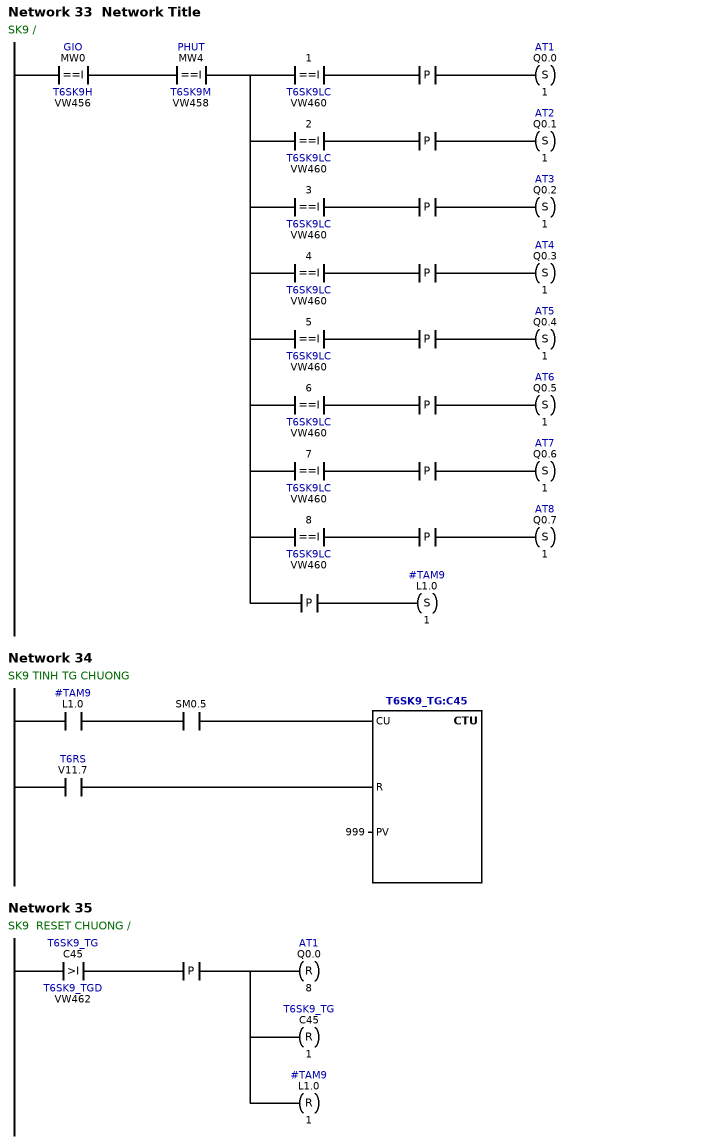
[picture p48: SBR7 networks 33-35]
Network 33 // Network Title
// SK9
// 	
LDW=   GIO:MW0, T6SK9H:VW456
AW=    PHUT:MW4, T6SK9M:VW458
LPS
AW=    1, T6SK9LC:VW460
EU
S      AT1:Q0.0, 1
LRD
AW=    2, T6SK9LC:VW460
EU
S      AT2:Q0.1, 1
LRD
AW=    3, T6SK9LC:VW460
EU
S      AT3:Q0.2, 1
LRD
AW=    4, T6SK9LC:VW460
EU
S      AT4:Q0.3, 1
LRD
AW=    5, T6SK9LC:VW460
EU
S      AT5:Q0.4, 1
LRD
AW=    6, T6SK9LC:VW460
EU
S      AT6:Q0.5, 1
LRD
AW=    7, T6SK9LC:VW460
EU
S      AT7:Q0.6, 1
LRD
AW=    8, T6SK9LC:VW460
EU
S      AT8:Q0.7, 1
LPP
EU
S      #TAM9:L1.0, 1
Network 34
// SK9 TINH TG CHUONG
LD     #TAM9:L1.0
A      SM0.5
LD     T6RS:V11.7
CTU    T6SK9_TG:C45, 999
Network 35
// SK9  RESET CHUONG
// 
LDW>   T6SK9_TG:C45, T6SK9_TGD:VW462
EU
R      AT1:Q0.0, 8
R      T6SK9_TG:C45, 1
R      #TAM9:L1.0, 1
Network 44 // Network Title
// Network Comment
Network 54 // Network Title
// Network Comment
Network 64 // Network Title
// Network Comment
Network 74 // Network Title
// Network Comment
END_SUBROUTINE_BLOCK

SUBROUTINE_BLOCK TH7:SBR8
TITLE=SUBROUTINE COMMENTS
VAR
TAM1:BOOL;	// L0.0 
TAM2:BOOL;	// L0.1 
TAM3:BOOL;	// L0.2 
TAM4:BOOL;	// L0.3 
TAM5:BOOL;	// L0.4 
TAM6:BOOL;	// L0.5 
TAM7:BOOL;	// L0.6 
TAM8:BOOL;	// L0.7 
TAM9:BOOL;	// L1.0 
END_VAR
BEGIN
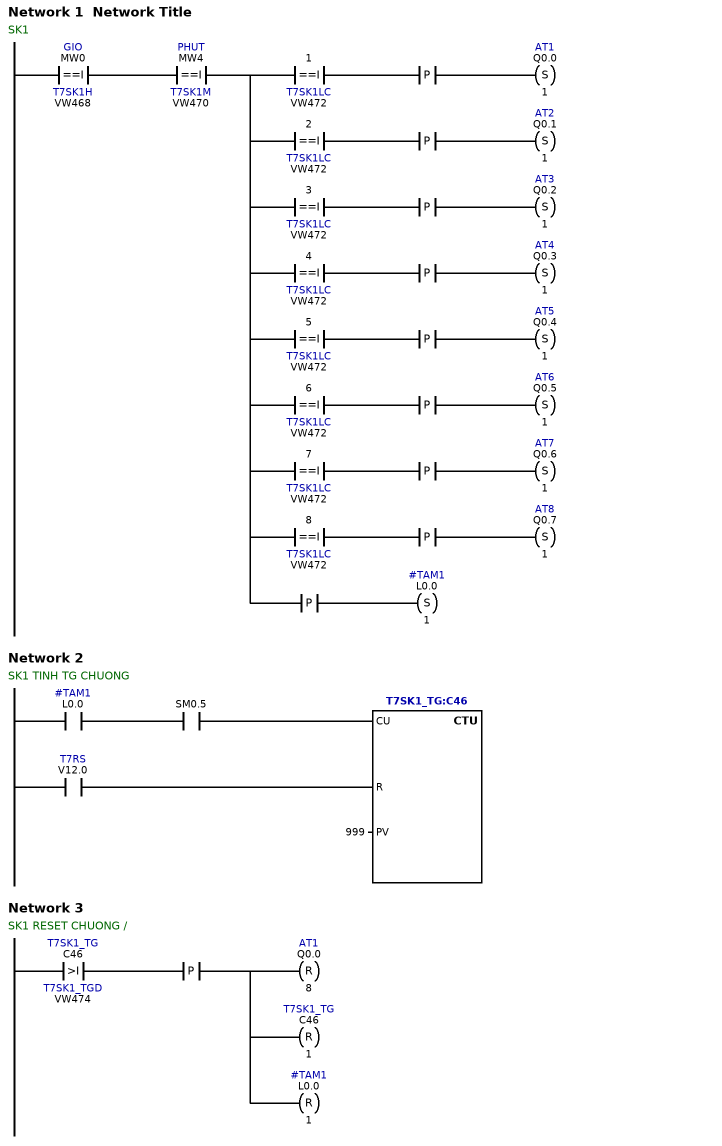
Network 1 // Network Title
// SK1	
LDW=   GIO:MW0, T7SK1H:VW468
AW=    PHUT:MW4, T7SK1M:VW470
LPS
AW=    1, T7SK1LC:VW472
EU
S      AT1:Q0.0, 1
LRD
AW=    2, T7SK1LC:VW472
EU
S      AT2:Q0.1, 1
LRD
AW=    3, T7SK1LC:VW472
EU
S      AT3:Q0.2, 1
LRD
AW=    4, T7SK1LC:VW472
EU
S      AT4:Q0.3, 1
LRD
AW=    5, T7SK1LC:VW472
EU
S      AT5:Q0.4, 1
LRD
AW=    6, T7SK1LC:VW472
EU
S      AT6:Q0.5, 1
LRD
AW=    7, T7SK1LC:VW472
EU
S      AT7:Q0.6, 1
LRD
AW=    8, T7SK1LC:VW472
EU
S      AT8:Q0.7, 1
LPP
EU
S      #TAM1:L0.0, 1
Network 2
// SK1 TINH TG CHUONG
LD     #TAM1:L0.0
A      SM0.5
LD     T7RS:V12.0
CTU    T7SK1_TG:C46, 999
Network 3
// SK1 RESET CHUONG
// 
LDW>   T7SK1_TG:C46, T7SK1_TGD:VW474
EU
R      AT1:Q0.0, 8
R      T7SK1_TG:C46, 1
R      #TAM1:L0.0, 1
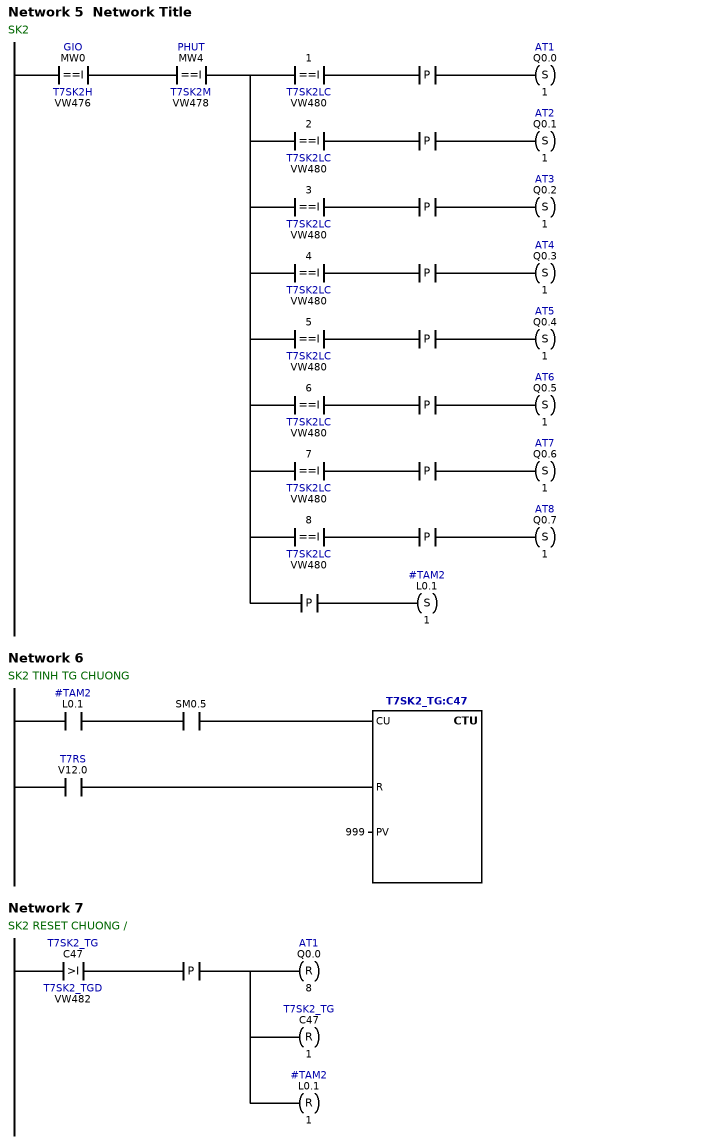
Network 5 // Network Title
// SK2
LDW=   GIO:MW0, T7SK2H:VW476
AW=    PHUT:MW4, T7SK2M:VW478
LPS
AW=    1, T7SK2LC:VW480
EU
S      AT1:Q0.0, 1
LRD
AW=    2, T7SK2LC:VW480
EU
S      AT2:Q0.1, 1
LRD
AW=    3, T7SK2LC:VW480
EU
S      AT3:Q0.2, 1
LRD
AW=    4, T7SK2LC:VW480
EU
S      AT4:Q0.3, 1
LRD
AW=    5, T7SK2LC:VW480
EU
S      AT5:Q0.4, 1
LRD
AW=    6, T7SK2LC:VW480
EU
S      AT6:Q0.5, 1
LRD
AW=    7, T7SK2LC:VW480
EU
S      AT7:Q0.6, 1
LRD
AW=    8, T7SK2LC:VW480
EU
S      AT8:Q0.7, 1
LPP
EU
S      #TAM2:L0.1, 1
Network 6
// SK2 TINH TG CHUONG
LD     #TAM2:L0.1
A      SM0.5
LD     T7RS:V12.0
CTU    T7SK2_TG:C47, 999
Network 7
// SK2 RESET CHUONG
// 
LDW>   T7SK2_TG:C47, T7SK2_TGD:VW482
EU
R      AT1:Q0.0, 8
R      T7SK2_TG:C47, 1
R      #TAM2:L0.1, 1
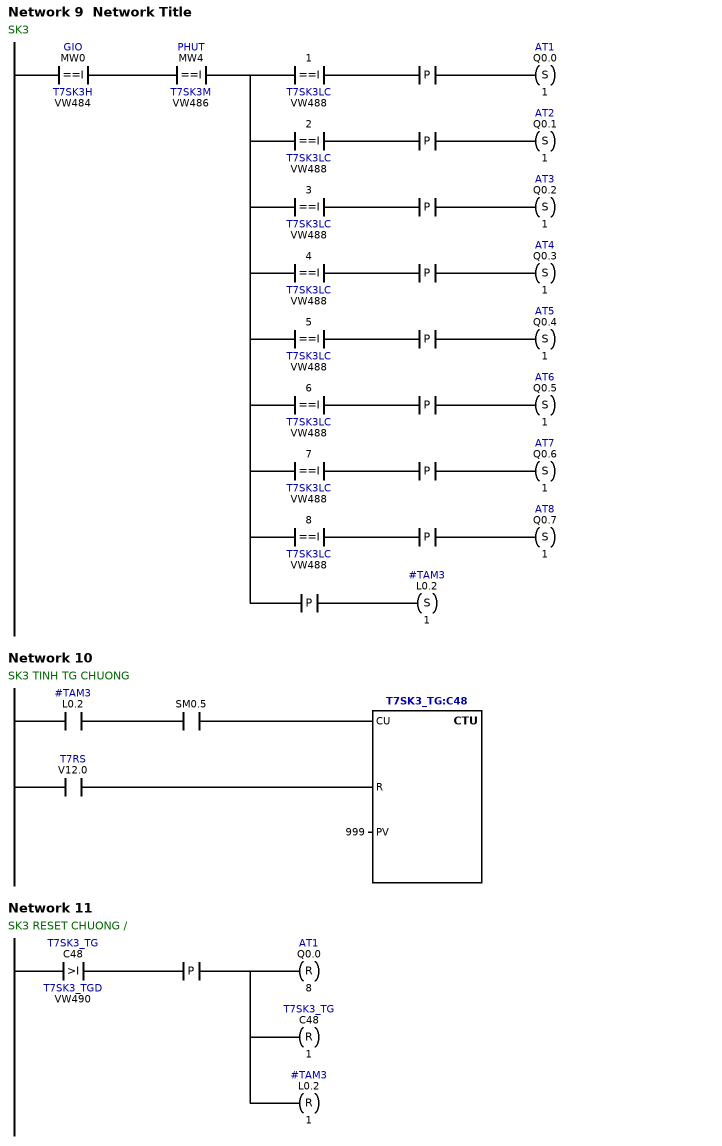
Network 9 // Network Title
// SK3	
LDW=   GIO:MW0, T7SK3H:VW484
AW=    PHUT:MW4, T7SK3M:VW486
LPS
AW=    1, T7SK3LC:VW488
EU
S      AT1:Q0.0, 1
LRD
AW=    2, T7SK3LC:VW488
EU
S      AT2:Q0.1, 1
LRD
AW=    3, T7SK3LC:VW488
EU
S      AT3:Q0.2, 1
LRD
AW=    4, T7SK3LC:VW488
EU
S      AT4:Q0.3, 1
LRD
AW=    5, T7SK3LC:VW488
EU
S      AT5:Q0.4, 1
LRD
AW=    6, T7SK3LC:VW488
EU
S      AT6:Q0.5, 1
LRD
AW=    7, T7SK3LC:VW488
EU
S      AT7:Q0.6, 1
LRD
AW=    8, T7SK3LC:VW488
EU
S      AT8:Q0.7, 1
LPP
EU
S      #TAM3:L0.2, 1
Network 10
// SK3 TINH TG CHUONG
LD     #TAM3:L0.2
A      SM0.5
LD     T7RS:V12.0
CTU    T7SK3_TG:C48, 999
Network 11
// SK3 RESET CHUONG
// 
LDW>   T7SK3_TG:C48, T7SK3_TGD:VW490
EU
R      AT1:Q0.0, 8
R      T7SK3_TG:C48, 1
R      #TAM3:L0.2, 1
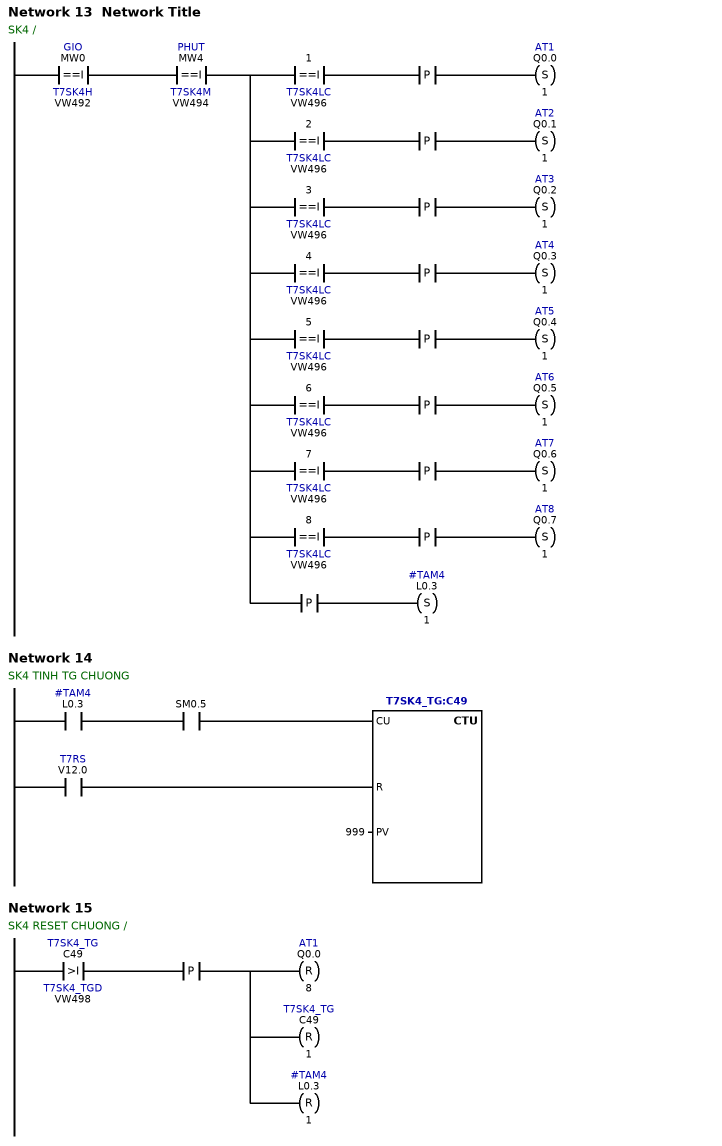
Network 13 // Network Title
// SK4
// 	
LDW=   GIO:MW0, T7SK4H:VW492
AW=    PHUT:MW4, T7SK4M:VW494
LPS
AW=    1, T7SK4LC:VW496
EU
S      AT1:Q0.0, 1
LRD
AW=    2, T7SK4LC:VW496
EU
S      AT2:Q0.1, 1
LRD
AW=    3, T7SK4LC:VW496
EU
S      AT3:Q0.2, 1
LRD
AW=    4, T7SK4LC:VW496
EU
S      AT4:Q0.3, 1
LRD
AW=    5, T7SK4LC:VW496
EU
S      AT5:Q0.4, 1
LRD
AW=    6, T7SK4LC:VW496
EU
S      AT6:Q0.5, 1
LRD
AW=    7, T7SK4LC:VW496
EU
S      AT7:Q0.6, 1
LRD
AW=    8, T7SK4LC:VW496
EU
S      AT8:Q0.7, 1
LPP
EU
S      #TAM4:L0.3, 1
Network 14
// SK4 TINH TG CHUONG
LD     #TAM4:L0.3
A      SM0.5
LD     T7RS:V12.0
CTU    T7SK4_TG:C49, 999
Network 15
// SK4 RESET CHUONG
// 
LDW>   T7SK4_TG:C49, T7SK4_TGD:VW498
EU
R      AT1:Q0.0, 8
R      T7SK4_TG:C49, 1
R      #TAM4:L0.3, 1
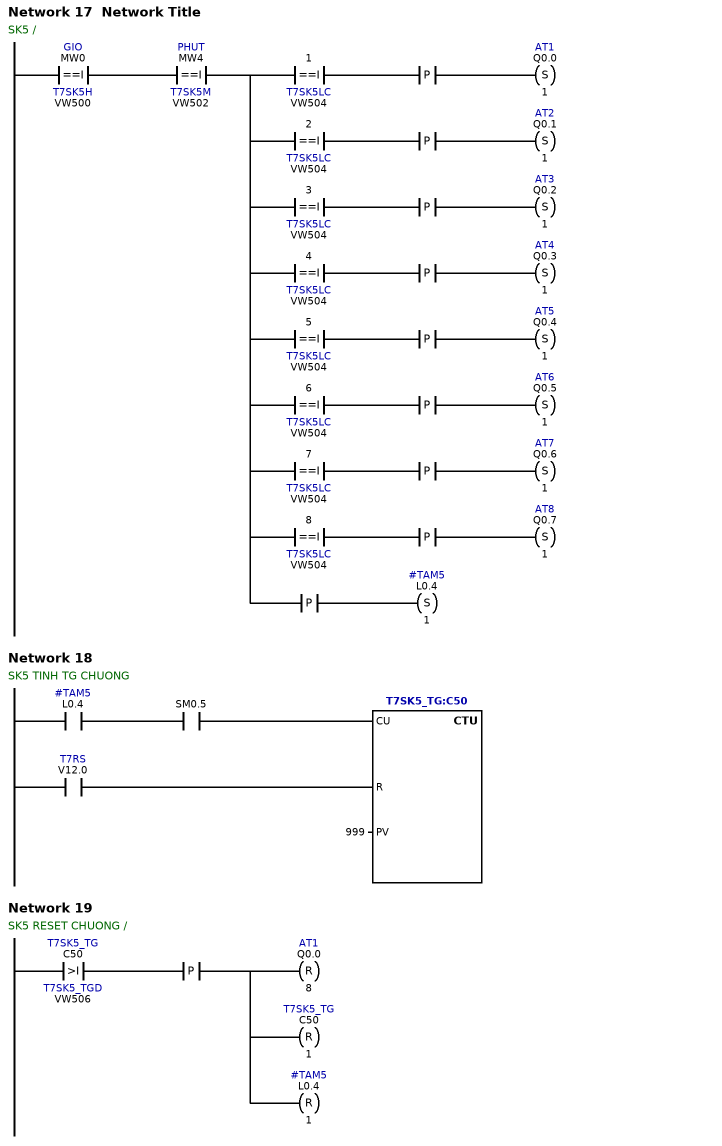
Network 17 // Network Title
// SK5
// 	
LDW=   GIO:MW0, T7SK5H:VW500
AW=    PHUT:MW4, T7SK5M:VW502
LPS
AW=    1, T7SK5LC:VW504
EU
S      AT1:Q0.0, 1
LRD
AW=    2, T7SK5LC:VW504
EU
S      AT2:Q0.1, 1
LRD
AW=    3, T7SK5LC:VW504
EU
S      AT3:Q0.2, 1
LRD
AW=    4, T7SK5LC:VW504
EU
S      AT4:Q0.3, 1
LRD
AW=    5, T7SK5LC:VW504
EU
S      AT5:Q0.4, 1
LRD
AW=    6, T7SK5LC:VW504
EU
S      AT6:Q0.5, 1
LRD
AW=    7, T7SK5LC:VW504
EU
S      AT7:Q0.6, 1
LRD
AW=    8, T7SK5LC:VW504
EU
S      AT8:Q0.7, 1
LPP
EU
S      #TAM5:L0.4, 1
Network 18
// SK5 TINH TG CHUONG
LD     #TAM5:L0.4
A      SM0.5
LD     T7RS:V12.0
CTU    T7SK5_TG:C50, 999
Network 19
// SK5 RESET CHUONG
// 
LDW>   T7SK5_TG:C50, T7SK5_TGD:VW506
EU
R      AT1:Q0.0, 8
R      T7SK5_TG:C50, 1
R      #TAM5:L0.4, 1
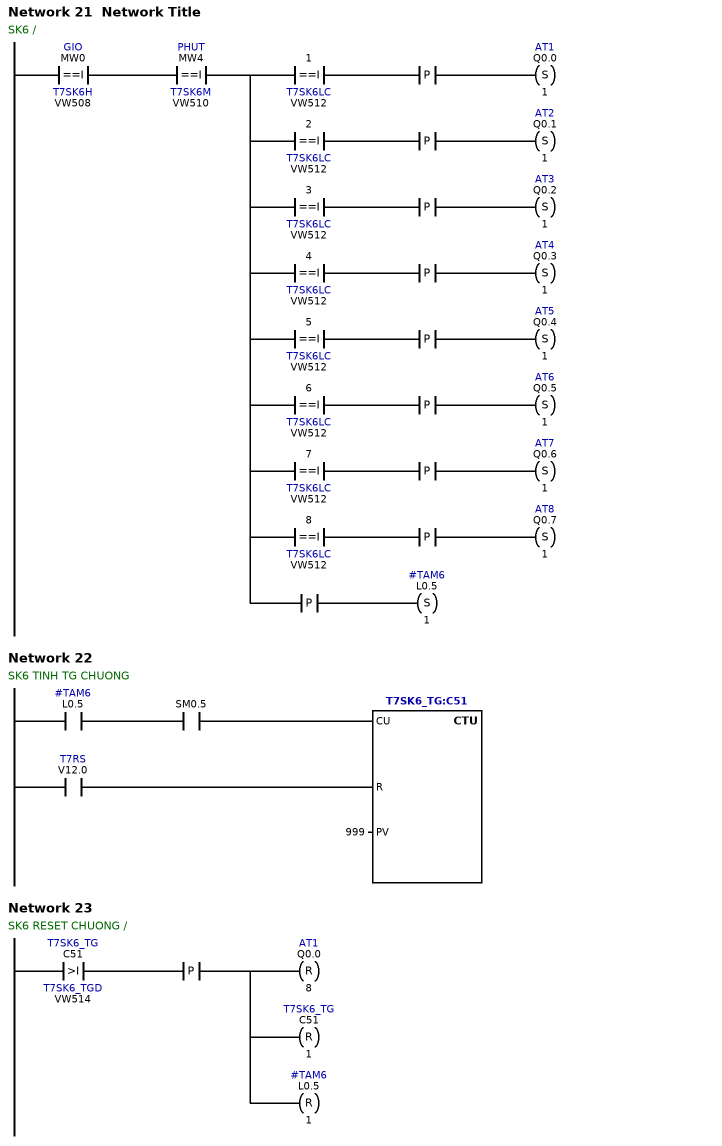
Network 21 // Network Title
// SK6
// 	
LDW=   GIO:MW0, T7SK6H:VW508
AW=    PHUT:MW4, T7SK6M:VW510
LPS
AW=    1, T7SK6LC:VW512
EU
S      AT1:Q0.0, 1
LRD
AW=    2, T7SK6LC:VW512
EU
S      AT2:Q0.1, 1
LRD
AW=    3, T7SK6LC:VW512
EU
S      AT3:Q0.2, 1
LRD
AW=    4, T7SK6LC:VW512
EU
S      AT4:Q0.3, 1
LRD
AW=    5, T7SK6LC:VW512
EU
S      AT5:Q0.4, 1
LRD
AW=    6, T7SK6LC:VW512
EU
S      AT6:Q0.5, 1
LRD
AW=    7, T7SK6LC:VW512
EU
S      AT7:Q0.6, 1
LRD
AW=    8, T7SK6LC:VW512
EU
S      AT8:Q0.7, 1
LPP
EU
S      #TAM6:L0.5, 1
Network 22
// SK6 TINH TG CHUONG
LD     #TAM6:L0.5
A      SM0.5
LD     T7RS:V12.0
CTU    T7SK6_TG:C51, 999
Network 23
// SK6 RESET CHUONG
// 
LDW>   T7SK6_TG:C51, T7SK6_TGD:VW514
EU
R      AT1:Q0.0, 8
R      T7SK6_TG:C51, 1
R      #TAM6:L0.5, 1
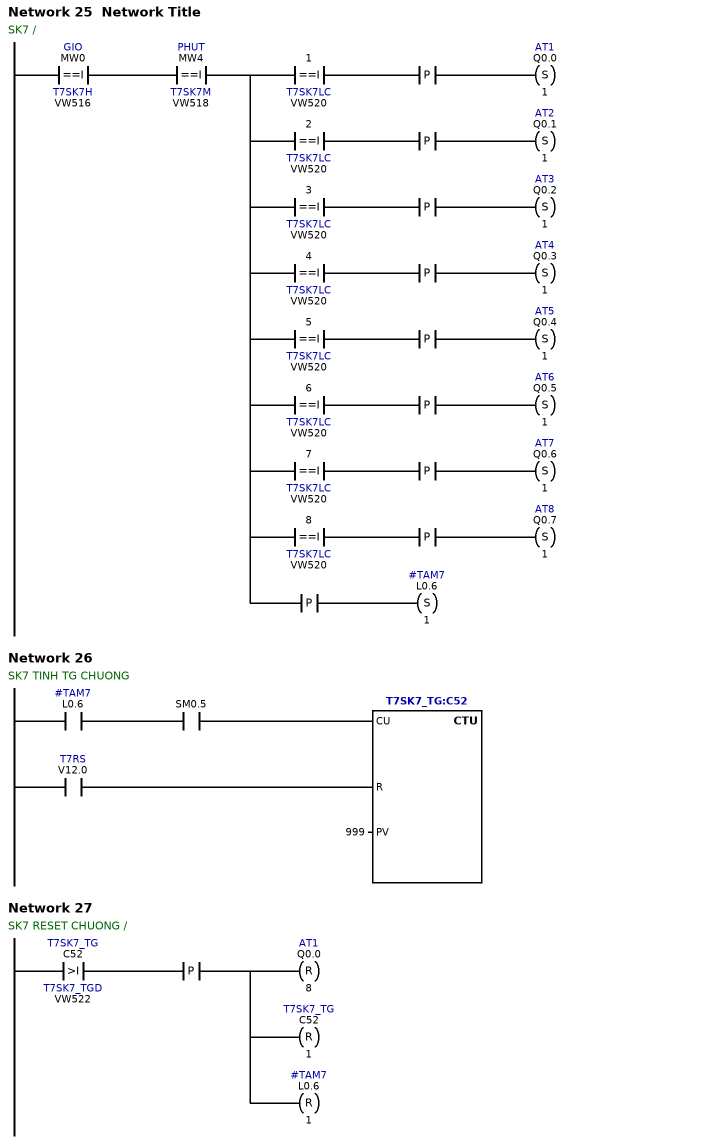
Network 25 // Network Title
// SK7
// 	
LDW=   GIO:MW0, T7SK7H:VW516
AW=    PHUT:MW4, T7SK7M:VW518
LPS
AW=    1, T7SK7LC:VW520
EU
S      AT1:Q0.0, 1
LRD
AW=    2, T7SK7LC:VW520
EU
S      AT2:Q0.1, 1
LRD
AW=    3, T7SK7LC:VW520
EU
S      AT3:Q0.2, 1
LRD
AW=    4, T7SK7LC:VW520
EU
S      AT4:Q0.3, 1
LRD
AW=    5, T7SK7LC:VW520
EU
S      AT5:Q0.4, 1
LRD
AW=    6, T7SK7LC:VW520
EU
S      AT6:Q0.5, 1
LRD
AW=    7, T7SK7LC:VW520
EU
S      AT7:Q0.6, 1
LRD
AW=    8, T7SK7LC:VW520
EU
S      AT8:Q0.7, 1
LPP
EU
S      #TAM7:L0.6, 1
Network 26
// SK7 TINH TG CHUONG
LD     #TAM7:L0.6
A      SM0.5
LD     T7RS:V12.0
CTU    T7SK7_TG:C52, 999
Network 27
// SK7 RESET CHUONG
// 
LDW>   T7SK7_TG:C52, T7SK7_TGD:VW522
EU
R      AT1:Q0.0, 8
R      T7SK7_TG:C52, 1
R      #TAM7:L0.6, 1
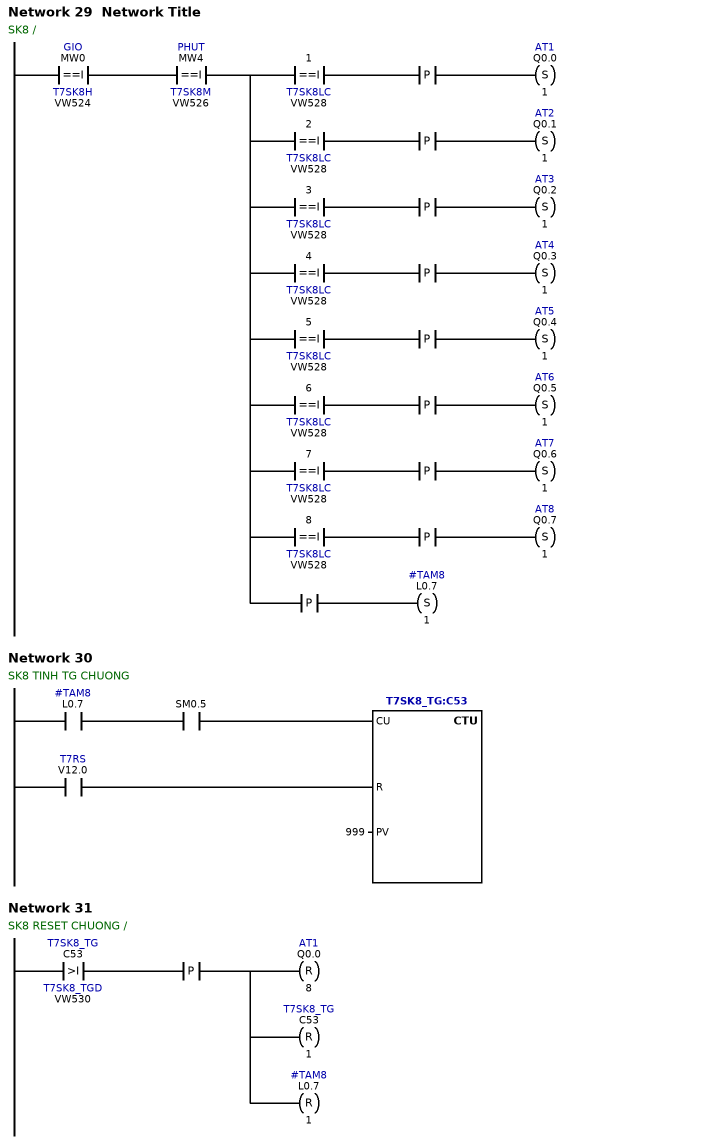
Network 29 // Network Title
// SK8
// 	
LDW=   GIO:MW0, T7SK8H:VW524
AW=    PHUT:MW4, T7SK8M:VW526
LPS
AW=    1, T7SK8LC:VW528
EU
S      AT1:Q0.0, 1
LRD
AW=    2, T7SK8LC:VW528
EU
S      AT2:Q0.1, 1
LRD
AW=    3, T7SK8LC:VW528
EU
S      AT3:Q0.2, 1
LRD
AW=    4, T7SK8LC:VW528
EU
S      AT4:Q0.3, 1
LRD
AW=    5, T7SK8LC:VW528
EU
S      AT5:Q0.4, 1
LRD
AW=    6, T7SK8LC:VW528
EU
S      AT6:Q0.5, 1
LRD
AW=    7, T7SK8LC:VW528
EU
S      AT7:Q0.6, 1
LRD
AW=    8, T7SK8LC:VW528
EU
S      AT8:Q0.7, 1
LPP
EU
S      #TAM8:L0.7, 1
Network 30
// SK8 TINH TG CHUONG
LD     #TAM8:L0.7
A      SM0.5
LD     T7RS:V12.0
CTU    T7SK8_TG:C53, 999
Network 31
// SK8 RESET CHUONG
// 
LDW>   T7SK8_TG:C53, T7SK8_TGD:VW530
EU
R      AT1:Q0.0, 8
R      T7SK8_TG:C53, 1
R      #TAM8:L0.7, 1
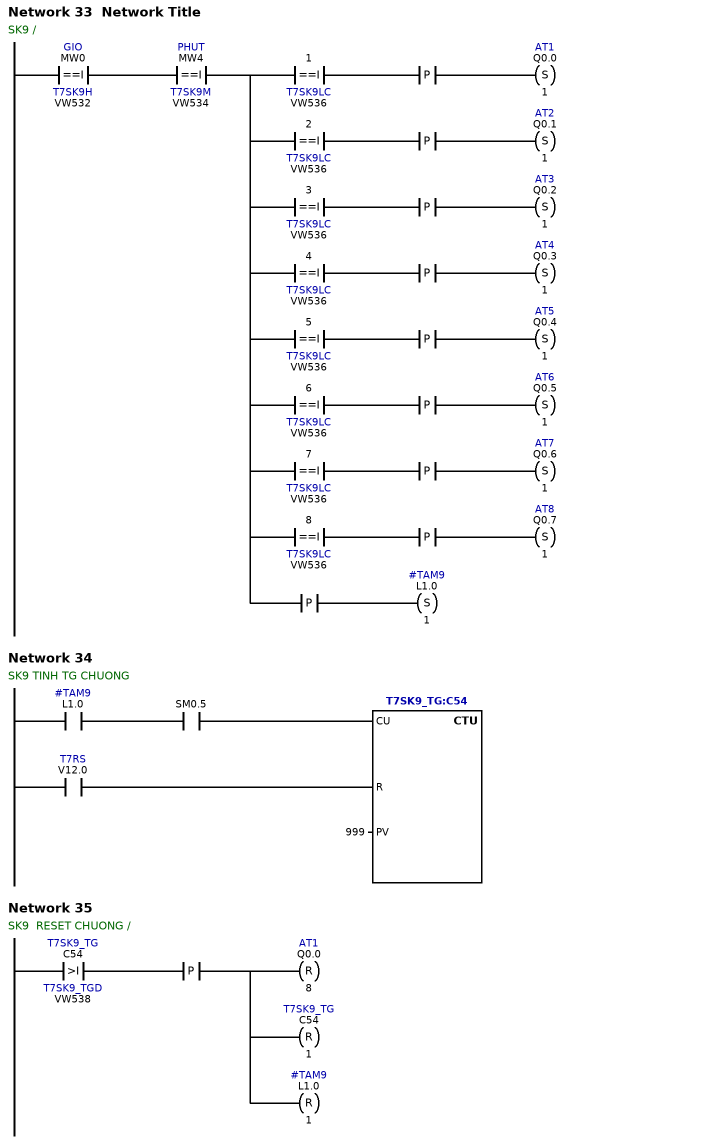
Network 33 // Network Title
// SK9
// 	
LDW=   GIO:MW0, T7SK9H:VW532
AW=    PHUT:MW4, T7SK9M:VW534
LPS
AW=    1, T7SK9LC:VW536
EU
S      AT1:Q0.0, 1
LRD
AW=    2, T7SK9LC:VW536
EU
S      AT2:Q0.1, 1
LRD
AW=    3, T7SK9LC:VW536
EU
S      AT3:Q0.2, 1
LRD
AW=    4, T7SK9LC:VW536
EU
S      AT4:Q0.3, 1
LRD
AW=    5, T7SK9LC:VW536
EU
S      AT5:Q0.4, 1
LRD
AW=    6, T7SK9LC:VW536
EU
S      AT6:Q0.5, 1
LRD
AW=    7, T7SK9LC:VW536
EU
S      AT7:Q0.6, 1
LRD
AW=    8, T7SK9LC:VW536
EU
S      AT8:Q0.7, 1
LPP
EU
S      #TAM9:L1.0, 1
Network 34
// SK9 TINH TG CHUONG
LD     #TAM9:L1.0
A      SM0.5
LD     T7RS:V12.0
CTU    T7SK9_TG:C54, 999
Network 35
// SK9  RESET CHUONG
// 
LDW>   T7SK9_TG:C54, T7SK9_TGD:VW538
EU
R      AT1:Q0.0, 8
R      T7SK9_TG:C54, 1
R      #TAM9:L1.0, 1
Network 44 // Network Title
// Network Comment
Network 54 // Network Title
// Network Comment
Network 64 // Network Title
// Network Comment
Network 74 // Network Title
// Network Comment
Network 84 // Network Title
// Network Comment
END_SUBROUTINE_BLOCK

SUBROUTINE_BLOCK CN:SBR9
TITLE=SUBROUTINE COMMENTS
VAR
TAM1:BOOL;	// L0.0 
TAM2:BOOL;	// L0.1 
TAM3:BOOL;	// L0.2 
TAM4:BOOL;	// L0.3 
TAM5:BOOL;	// L0.4 
TAM6:BOOL;	// L0.5 
TAM7:BOOL;	// L0.6 
TAM8:BOOL;	// L0.7 
TAM9:BOOL;	// L1.0 
END_VAR
BEGIN
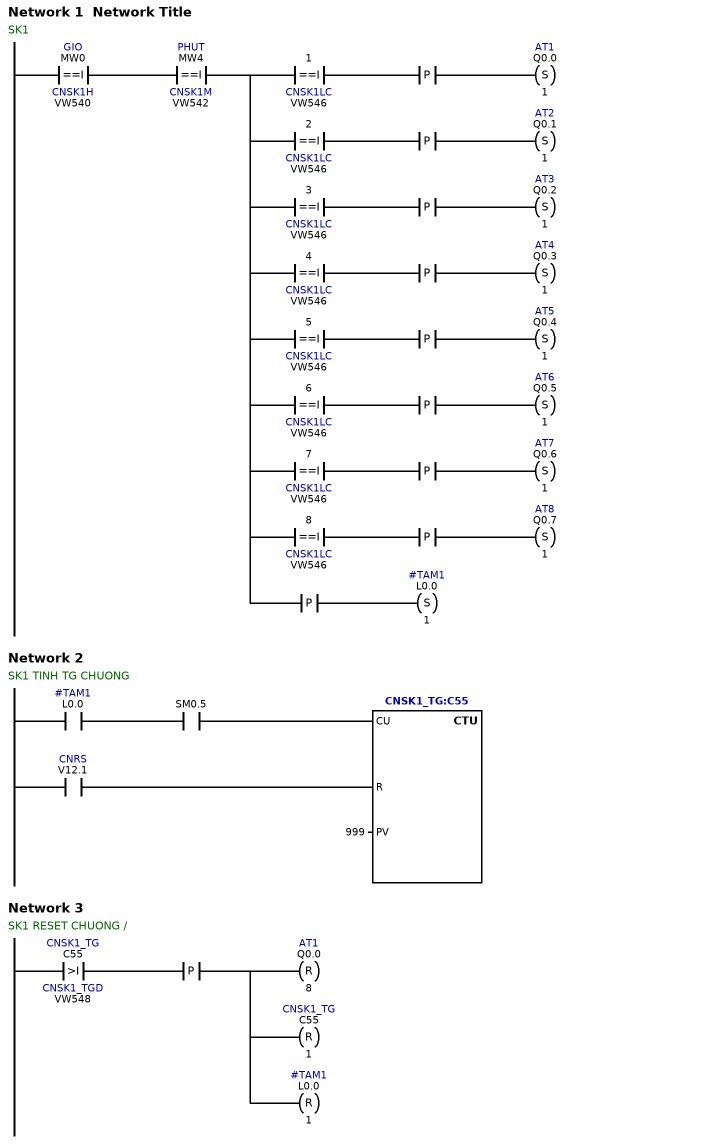
Network 1 // Network Title
// SK1	
LDW=   GIO:MW0, CNSK1H:VW540
AW=    PHUT:MW4, CNSK1M:VW542
LPS
AW=    1, CNSK1LC:VW546
EU
S      AT1:Q0.0, 1
LRD
AW=    2, CNSK1LC:VW546
EU
S      AT2:Q0.1, 1
LRD
AW=    3, CNSK1LC:VW546
EU
S      AT3:Q0.2, 1
LRD
AW=    4, CNSK1LC:VW546
EU
S      AT4:Q0.3, 1
LRD
AW=    5, CNSK1LC:VW546
EU
S      AT5:Q0.4, 1
LRD
AW=    6, CNSK1LC:VW546
EU
S      AT6:Q0.5, 1
LRD
AW=    7, CNSK1LC:VW546
EU
S      AT7:Q0.6, 1
LRD
AW=    8, CNSK1LC:VW546
EU
S      AT8:Q0.7, 1
LPP
EU
S      #TAM1:L0.0, 1
Network 2
// SK1 TINH TG CHUONG
LD     #TAM1:L0.0
A      SM0.5
LD     CNRS:V12.1
CTU    CNSK1_TG:C55, 999
Network 3
// SK1 RESET CHUONG
// 
LDW>   CNSK1_TG:C55, CNSK1_TGD:VW548
EU
R      AT1:Q0.0, 8
R      CNSK1_TG:C55, 1
R      #TAM1:L0.0, 1
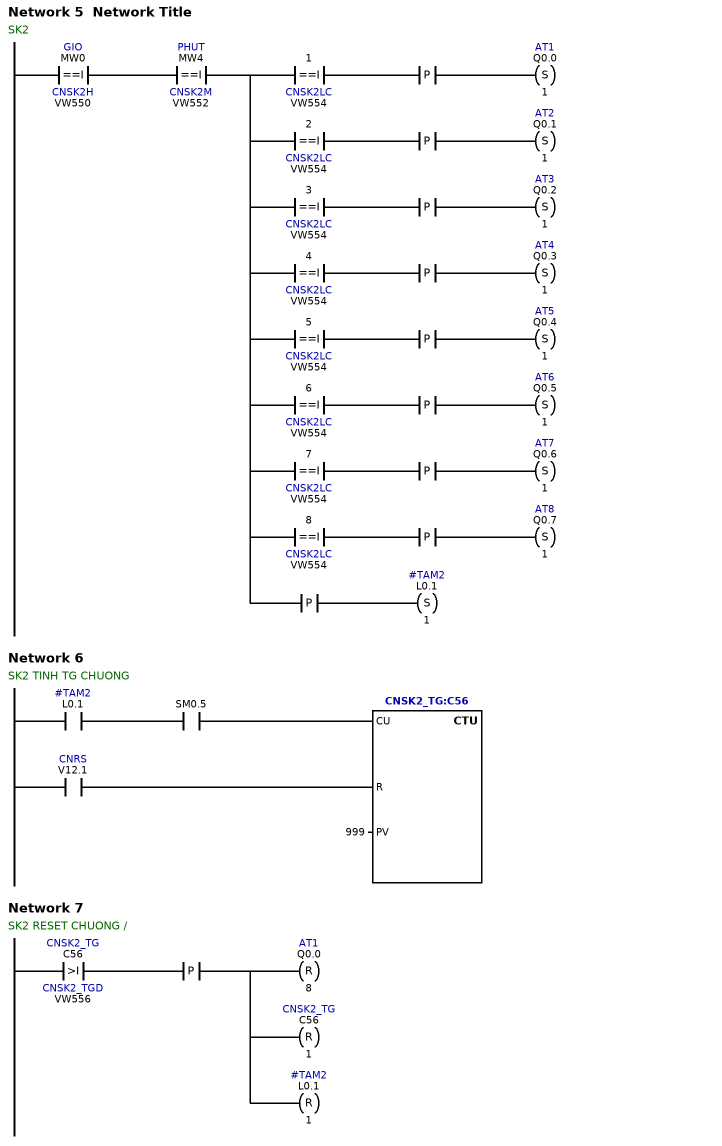
Network 5 // Network Title
// SK2
LDW=   GIO:MW0, CNSK2H:VW550
AW=    PHUT:MW4, CNSK2M:VW552
LPS
AW=    1, CNSK2LC:VW554
EU
S      AT1:Q0.0, 1
LRD
AW=    2, CNSK2LC:VW554
EU
S      AT2:Q0.1, 1
LRD
AW=    3, CNSK2LC:VW554
EU
S      AT3:Q0.2, 1
LRD
AW=    4, CNSK2LC:VW554
EU
S      AT4:Q0.3, 1
LRD
AW=    5, CNSK2LC:VW554
EU
S      AT5:Q0.4, 1
LRD
AW=    6, CNSK2LC:VW554
EU
S      AT6:Q0.5, 1
LRD
AW=    7, CNSK2LC:VW554
EU
S      AT7:Q0.6, 1
LRD
AW=    8, CNSK2LC:VW554
EU
S      AT8:Q0.7, 1
LPP
EU
S      #TAM2:L0.1, 1
Network 6
// SK2 TINH TG CHUONG
LD     #TAM2:L0.1
A      SM0.5
LD     CNRS:V12.1
CTU    CNSK2_TG:C56, 999
Network 7
// SK2 RESET CHUONG
// 
LDW>   CNSK2_TG:C56, CNSK2_TGD:VW556
EU
R      AT1:Q0.0, 8
R      CNSK2_TG:C56, 1
R      #TAM2:L0.1, 1
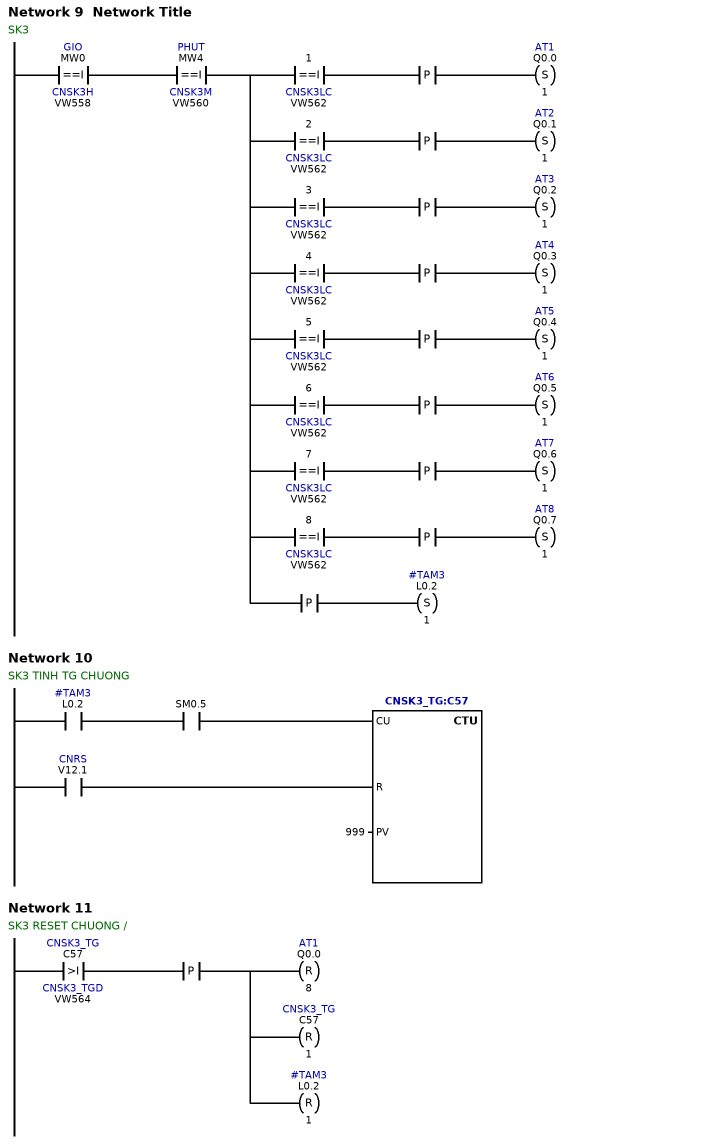
Network 9 // Network Title
// SK3	
LDW=   GIO:MW0, CNSK3H:VW558
AW=    PHUT:MW4, CNSK3M:VW560
LPS
AW=    1, CNSK3LC:VW562
EU
S      AT1:Q0.0, 1
LRD
AW=    2, CNSK3LC:VW562
EU
S      AT2:Q0.1, 1
LRD
AW=    3, CNSK3LC:VW562
EU
S      AT3:Q0.2, 1
LRD
AW=    4, CNSK3LC:VW562
EU
S      AT4:Q0.3, 1
LRD
AW=    5, CNSK3LC:VW562
EU
S      AT5:Q0.4, 1
LRD
AW=    6, CNSK3LC:VW562
EU
S      AT6:Q0.5, 1
LRD
AW=    7, CNSK3LC:VW562
EU
S      AT7:Q0.6, 1
LRD
AW=    8, CNSK3LC:VW562
EU
S      AT8:Q0.7, 1
LPP
EU
S      #TAM3:L0.2, 1
Network 10
// SK3 TINH TG CHUONG
LD     #TAM3:L0.2
A      SM0.5
LD     CNRS:V12.1
CTU    CNSK3_TG:C57, 999
Network 11
// SK3 RESET CHUONG
// 
LDW>   CNSK3_TG:C57, CNSK3_TGD:VW564
EU
R      AT1:Q0.0, 8
R      CNSK3_TG:C57, 1
R      #TAM3:L0.2, 1
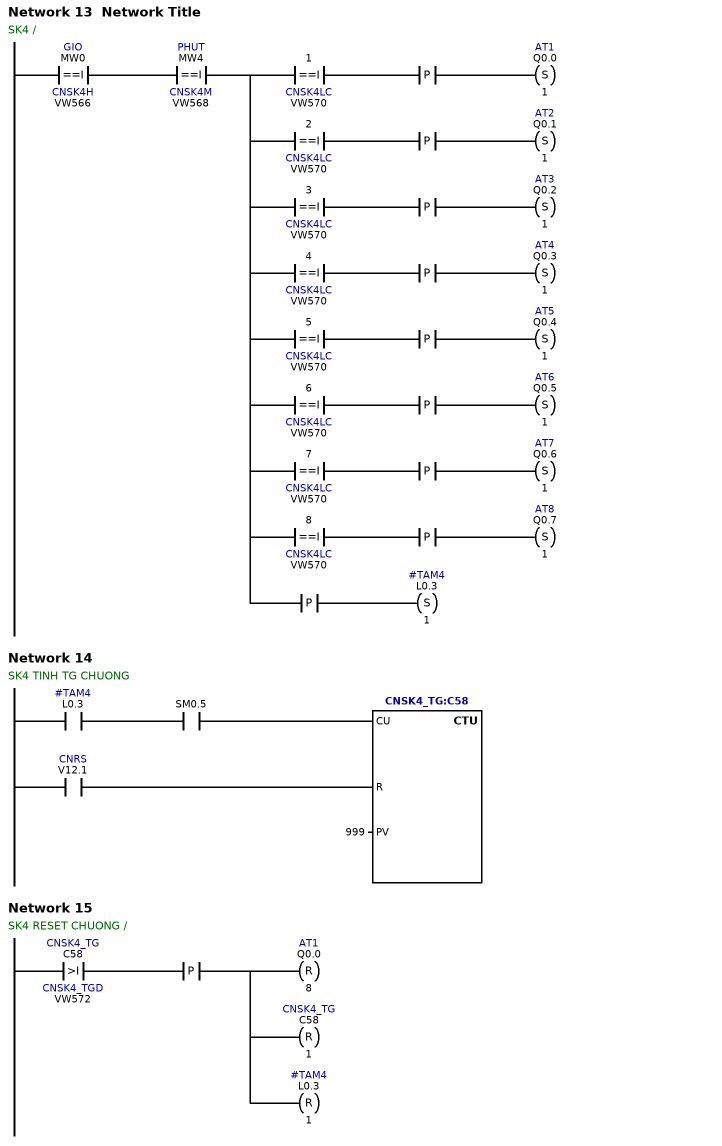
Network 13 // Network Title
// SK4
// 	
LDW=   GIO:MW0, CNSK4H:VW566
AW=    PHUT:MW4, CNSK4M:VW568
LPS
AW=    1, CNSK4LC:VW570
EU
S      AT1:Q0.0, 1
LRD
AW=    2, CNSK4LC:VW570
EU
S      AT2:Q0.1, 1
LRD
AW=    3, CNSK4LC:VW570
EU
S      AT3:Q0.2, 1
LRD
AW=    4, CNSK4LC:VW570
EU
S      AT4:Q0.3, 1
LRD
AW=    5, CNSK4LC:VW570
EU
S      AT5:Q0.4, 1
LRD
AW=    6, CNSK4LC:VW570
EU
S      AT6:Q0.5, 1
LRD
AW=    7, CNSK4LC:VW570
EU
S      AT7:Q0.6, 1
LRD
AW=    8, CNSK4LC:VW570
EU
S      AT8:Q0.7, 1
LPP
EU
S      #TAM4:L0.3, 1
Network 14
// SK4 TINH TG CHUONG
LD     #TAM4:L0.3
A      SM0.5
LD     CNRS:V12.1
CTU    CNSK4_TG:C58, 999
Network 15
// SK4 RESET CHUONG
// 
LDW>   CNSK4_TG:C58, CNSK4_TGD:VW572
EU
R      AT1:Q0.0, 8
R      CNSK4_TG:C58, 1
R      #TAM4:L0.3, 1
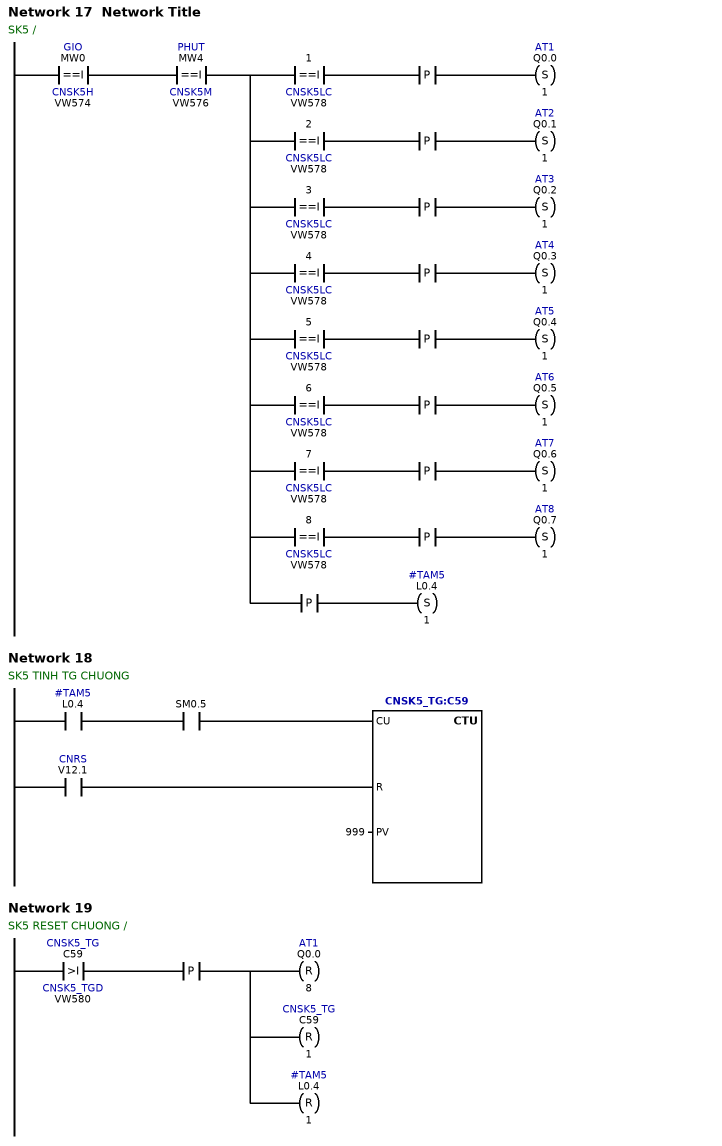
Network 17 // Network Title
// SK5
// 	
LDW=   GIO:MW0, CNSK5H:VW574
AW=    PHUT:MW4, CNSK5M:VW576
LPS
AW=    1, CNSK5LC:VW578
EU
S      AT1:Q0.0, 1
LRD
AW=    2, CNSK5LC:VW578
EU
S      AT2:Q0.1, 1
LRD
AW=    3, CNSK5LC:VW578
EU
S      AT3:Q0.2, 1
LRD
AW=    4, CNSK5LC:VW578
EU
S      AT4:Q0.3, 1
LRD
AW=    5, CNSK5LC:VW578
EU
S      AT5:Q0.4, 1
LRD
AW=    6, CNSK5LC:VW578
EU
S      AT6:Q0.5, 1
LRD
AW=    7, CNSK5LC:VW578
EU
S      AT7:Q0.6, 1
LRD
AW=    8, CNSK5LC:VW578
EU
S      AT8:Q0.7, 1
LPP
EU
S      #TAM5:L0.4, 1
Network 18
// SK5 TINH TG CHUONG
LD     #TAM5:L0.4
A      SM0.5
LD     CNRS:V12.1
CTU    CNSK5_TG:C59, 999
Network 19
// SK5 RESET CHUONG
// 
LDW>   CNSK5_TG:C59, CNSK5_TGD:VW580
EU
R      AT1:Q0.0, 8
R      CNSK5_TG:C59, 1
R      #TAM5:L0.4, 1
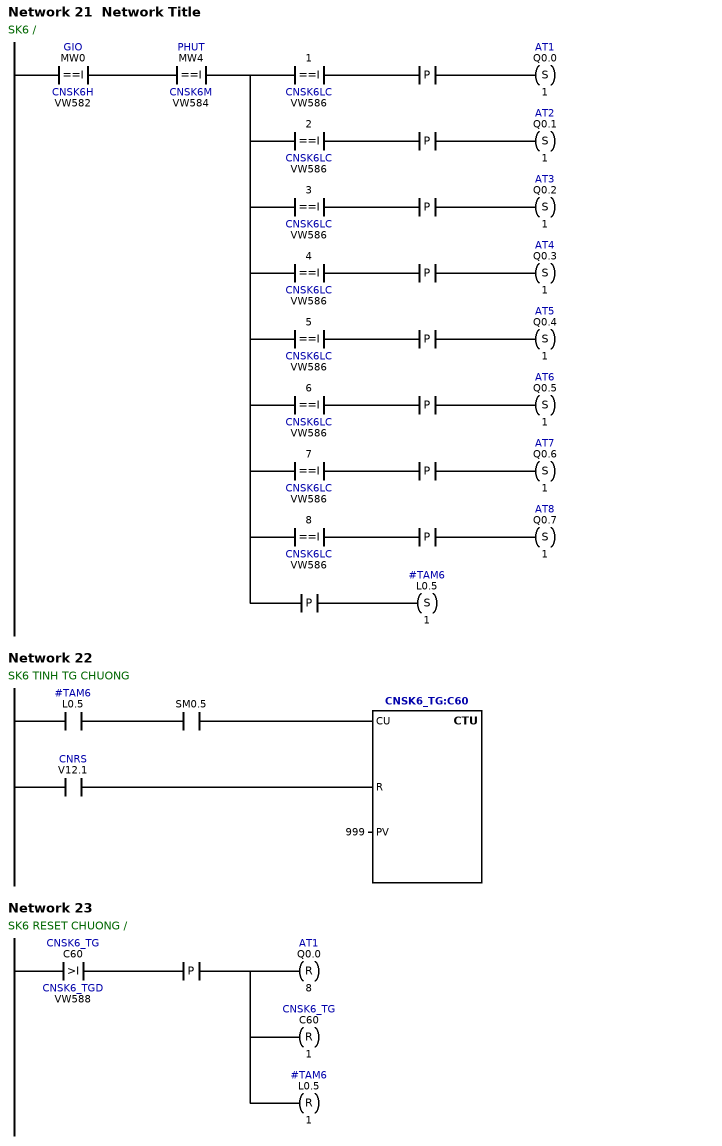
Network 21 // Network Title
// SK6
// 	
LDW=   GIO:MW0, CNSK6H:VW582
AW=    PHUT:MW4, CNSK6M:VW584
LPS
AW=    1, CNSK6LC:VW586
EU
S      AT1:Q0.0, 1
LRD
AW=    2, CNSK6LC:VW586
EU
S      AT2:Q0.1, 1
LRD
AW=    3, CNSK6LC:VW586
EU
S      AT3:Q0.2, 1
LRD
AW=    4, CNSK6LC:VW586
EU
S      AT4:Q0.3, 1
LRD
AW=    5, CNSK6LC:VW586
EU
S      AT5:Q0.4, 1
LRD
AW=    6, CNSK6LC:VW586
EU
S      AT6:Q0.5, 1
LRD
AW=    7, CNSK6LC:VW586
EU
S      AT7:Q0.6, 1
LRD
AW=    8, CNSK6LC:VW586
EU
S      AT8:Q0.7, 1
LPP
EU
S      #TAM6:L0.5, 1
Network 22
// SK6 TINH TG CHUONG
LD     #TAM6:L0.5
A      SM0.5
LD     CNRS:V12.1
CTU    CNSK6_TG:C60, 999
Network 23
// SK6 RESET CHUONG
// 
LDW>   CNSK6_TG:C60, CNSK6_TGD:VW588
EU
R      AT1:Q0.0, 8
R      CNSK6_TG:C60, 1
R      #TAM6:L0.5, 1
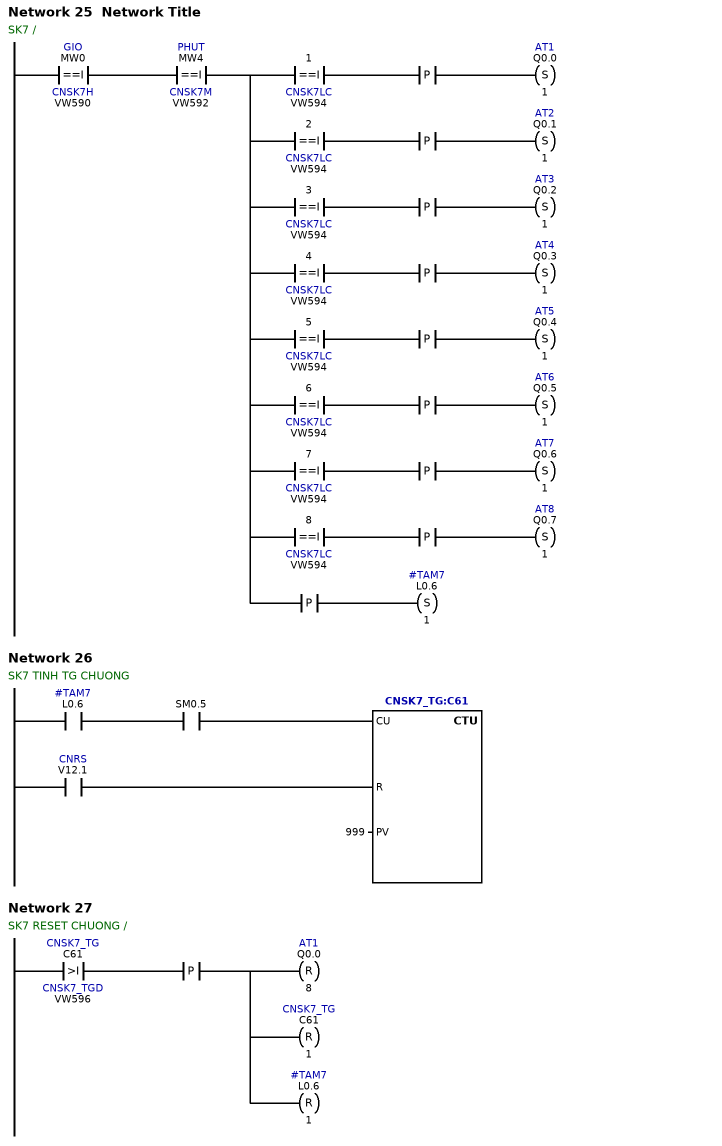
Network 25 // Network Title
// SK7
// 	
LDW=   GIO:MW0, CNSK7H:VW590
AW=    PHUT:MW4, CNSK7M:VW592
LPS
AW=    1, CNSK7LC:VW594
EU
S      AT1:Q0.0, 1
LRD
AW=    2, CNSK7LC:VW594
EU
S      AT2:Q0.1, 1
LRD
AW=    3, CNSK7LC:VW594
EU
S      AT3:Q0.2, 1
LRD
AW=    4, CNSK7LC:VW594
EU
S      AT4:Q0.3, 1
LRD
AW=    5, CNSK7LC:VW594
EU
S      AT5:Q0.4, 1
LRD
AW=    6, CNSK7LC:VW594
EU
S      AT6:Q0.5, 1
LRD
AW=    7, CNSK7LC:VW594
EU
S      AT7:Q0.6, 1
LRD
AW=    8, CNSK7LC:VW594
EU
S      AT8:Q0.7, 1
LPP
EU
S      #TAM7:L0.6, 1
Network 26
// SK7 TINH TG CHUONG
LD     #TAM7:L0.6
A      SM0.5
LD     CNRS:V12.1
CTU    CNSK7_TG:C61, 999
Network 27
// SK7 RESET CHUONG
// 
LDW>   CNSK7_TG:C61, CNSK7_TGD:VW596
EU
R      AT1:Q0.0, 8
R      CNSK7_TG:C61, 1
R      #TAM7:L0.6, 1
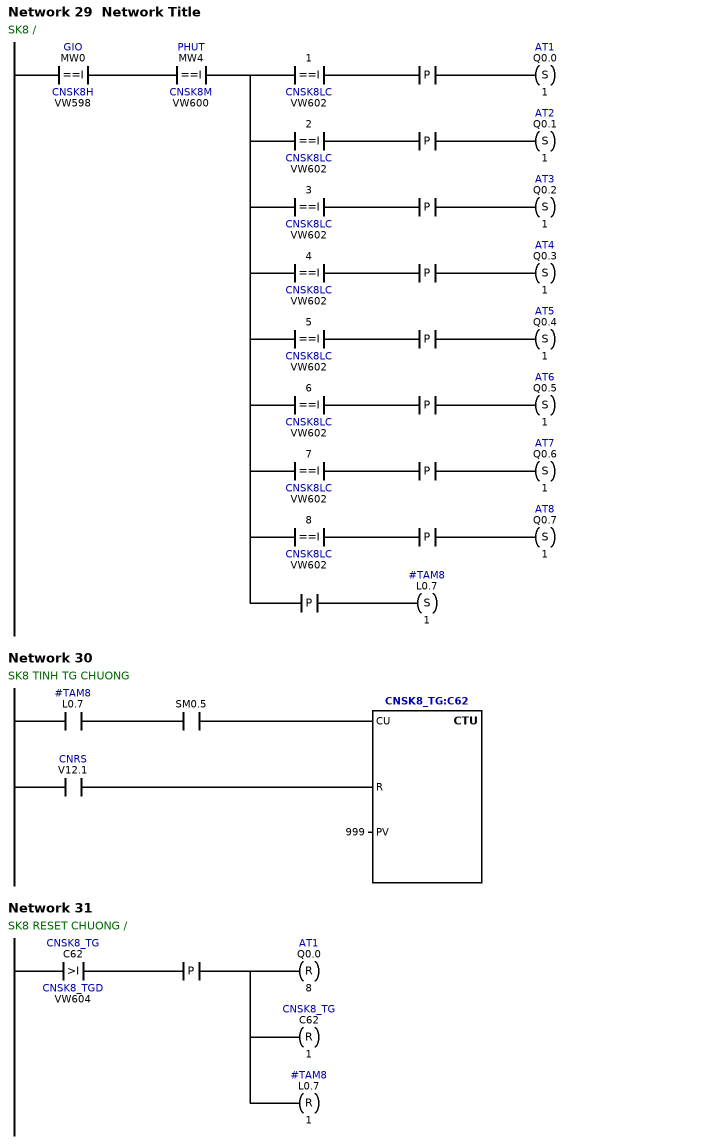
Network 29 // Network Title
// SK8
// 	
LDW=   GIO:MW0, CNSK8H:VW598
AW=    PHUT:MW4, CNSK8M:VW600
LPS
AW=    1, CNSK8LC:VW602
EU
S      AT1:Q0.0, 1
LRD
AW=    2, CNSK8LC:VW602
EU
S      AT2:Q0.1, 1
LRD
AW=    3, CNSK8LC:VW602
EU
S      AT3:Q0.2, 1
LRD
AW=    4, CNSK8LC:VW602
EU
S      AT4:Q0.3, 1
LRD
AW=    5, CNSK8LC:VW602
EU
S      AT5:Q0.4, 1
LRD
AW=    6, CNSK8LC:VW602
EU
S      AT6:Q0.5, 1
LRD
AW=    7, CNSK8LC:VW602
EU
S      AT7:Q0.6, 1
LRD
AW=    8, CNSK8LC:VW602
EU
S      AT8:Q0.7, 1
LPP
EU
S      #TAM8:L0.7, 1
Network 30
// SK8 TINH TG CHUONG
LD     #TAM8:L0.7
A      SM0.5
LD     CNRS:V12.1
CTU    CNSK8_TG:C62, 999
Network 31
// SK8 RESET CHUONG
// 
LDW>   CNSK8_TG:C62, CNSK8_TGD:VW604
EU
R      AT1:Q0.0, 8
R      CNSK8_TG:C62, 1
R      #TAM8:L0.7, 1
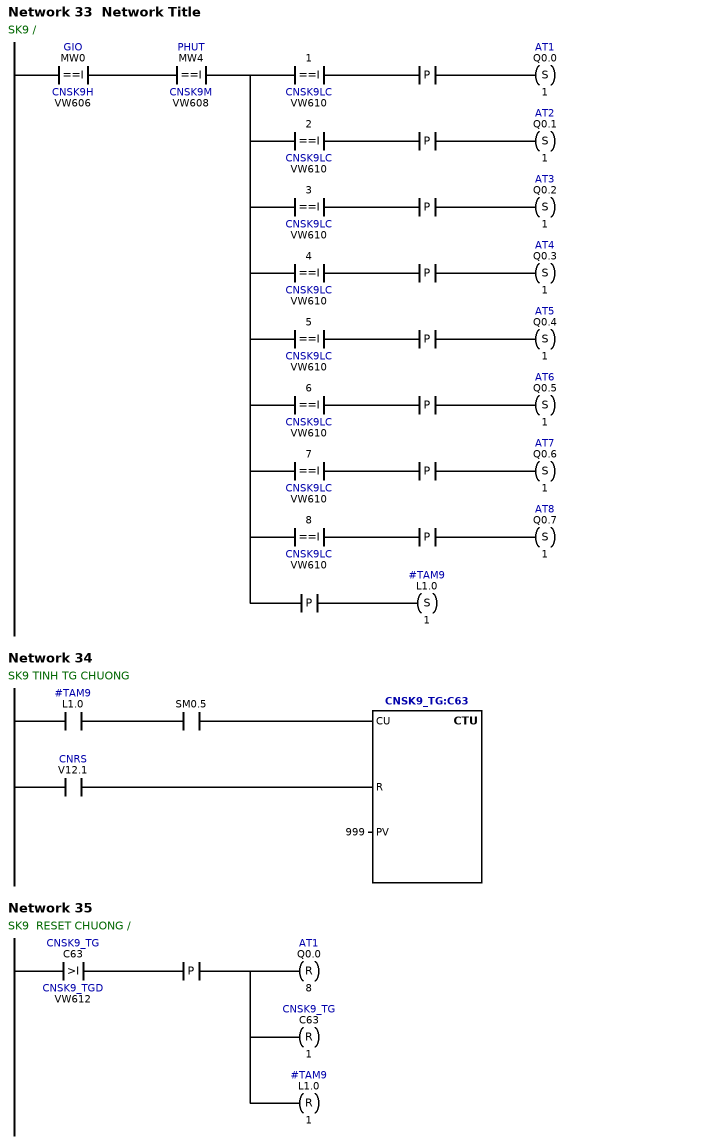
Network 33 // Network Title
// SK9
// 	
LDW=   GIO:MW0, CNSK9H:VW606
AW=    PHUT:MW4, CNSK9M:VW608
LPS
AW=    1, CNSK9LC:VW610
EU
S      AT1:Q0.0, 1
LRD
AW=    2, CNSK9LC:VW610
EU
S      AT2:Q0.1, 1
LRD
AW=    3, CNSK9LC:VW610
EU
S      AT3:Q0.2, 1
LRD
AW=    4, CNSK9LC:VW610
EU
S      AT4:Q0.3, 1
LRD
AW=    5, CNSK9LC:VW610
EU
S      AT5:Q0.4, 1
LRD
AW=    6, CNSK9LC:VW610
EU
S      AT6:Q0.5, 1
LRD
AW=    7, CNSK9LC:VW610
EU
S      AT7:Q0.6, 1
LRD
AW=    8, CNSK9LC:VW610
EU
S      AT8:Q0.7, 1
LPP
EU
S      #TAM9:L1.0, 1
Network 34
// SK9 TINH TG CHUONG
LD     #TAM9:L1.0
A      SM0.5
LD     CNRS:V12.1
CTU    CNSK9_TG:C63, 999
Network 35
// SK9  RESET CHUONG
// 
LDW>   CNSK9_TG:C63, CNSK9_TGD:VW612
EU
R      AT1:Q0.0, 8
R      CNSK9_TG:C63, 1
R      #TAM9:L1.0, 1
Network 44 // Network Title
// Network Comment
Network 54 // Network Title
// Network Comment
Network 64 // Network Title
// Network Comment
Network 74 // Network Title
// Network Comment
Network 84 // Network Title
// Network Comment
Network 94 // Network Title
// Network Comment
END_SUBROUTINE_BLOCK
